FUNCTION_BLOCK ADD_112C76C471B7A99C2 (* Add *)
  (* Standard: 61499-2 *)
  (* Version 1.1, 24.06.2019, winkhub, nxtControl GmbH, support TIME *)
  PACKAGE UAO.Hackathon;
  (* Compiler Cpp *)
  {SET_ATTRIBUTE(Runtime.FBType.ImplementingType, Runtime.Standard#DYNGEN_ADD)}
  {SET_ATTRIBUTE(Configuration.GenericFBType.InterfaceParams, Runtime.Standard#CNT:=2;IN${CNT$}:DINT)}
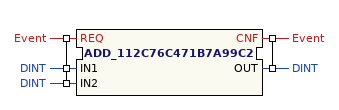
  EVENT_INPUT
    REQ WITH IN1, IN2; (* Normal Execution Request *)
  END_EVENT
  EVENT_OUTPUT
    CNF WITH OUT; (* Execution Confirmation *)
  END_EVENT
  VAR_INPUT
    IN1 : DINT; (* Argument *)
    IN2 : DINT; (* Argument *)
  END_VAR
  VAR_OUTPUT
    OUT : DINT; (* Result: IN1 + IN2 + ... *)
  END_VAR
  EC_STATES
    START;
  END_STATES
END_FUNCTION_BLOCK
